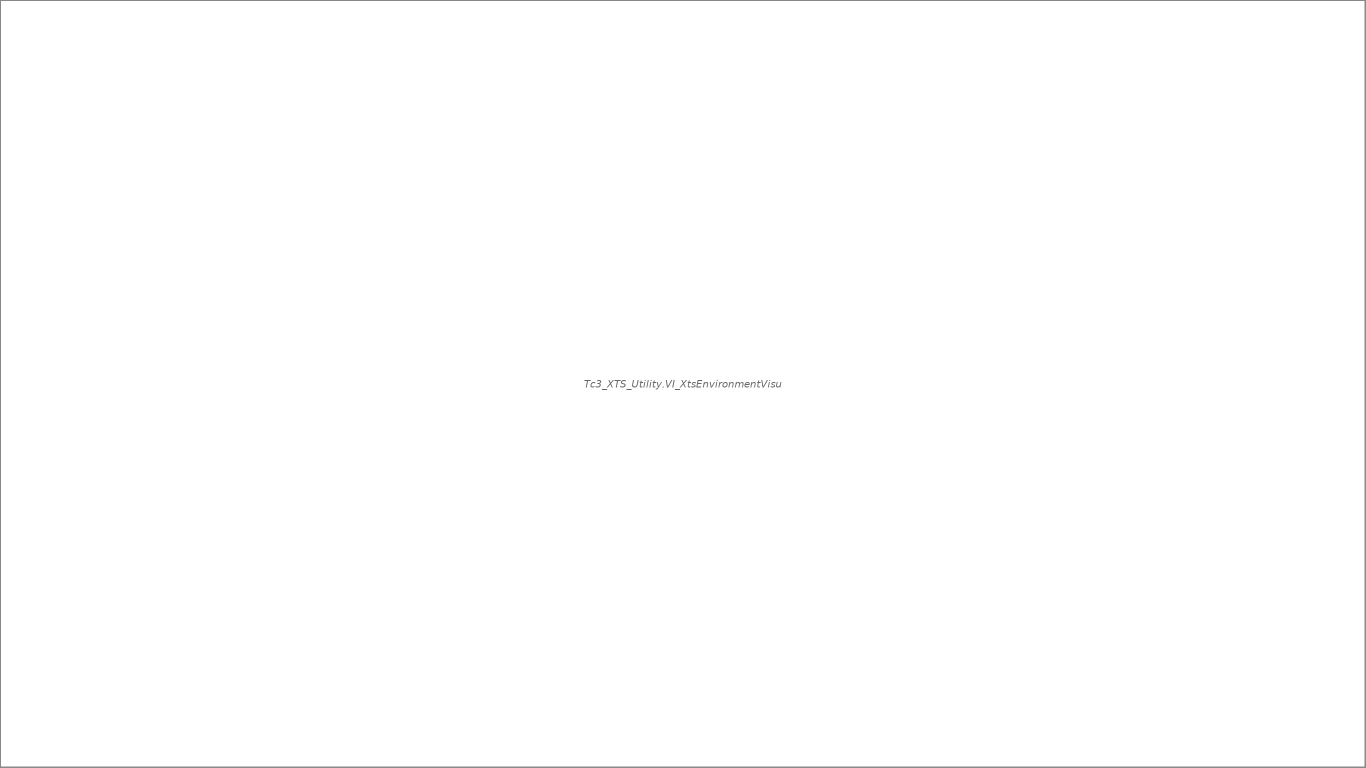
VISUALIZATION DiagnosticVisu  // 1366x768
    Frame (0,0 1366x768)
        shows Tc3_XTS_Utility.VI_XtsEnvironmentVisu()
END_VISUALIZATION

(* stored: Version 1.1.0.1, ProductVersion 3.1.4024.12
   Visu DiagnosticVisu: Id {0a14cc89-148e-0392-1f20-d50acac1a592} *)
